INTERFACE I_SnappySetupConfigSerializer

METHOD UseSerializer : I_SnappySetupConfigBuild
VAR_INPUT
	itfSerializer	: I_Serializer;
END_VAR
END_METHOD

END_INTERFACE

(* stored: Version 1.1.0.1, ProductVersion 3.1.4026.18
   Itf I_SnappySetupConfigSerializer: Id {edd9672f-1e06-4a2e-b72e-ed58d685e531}
   Method UseSerializer: Id {d78d7c7d-a03a-481b-9a0c-f9fc721210f4} *)
